Fanuc KAREL source: MSG_DISCO.kl

PROGRAM T
%NOLOCKGROUP
VAR
 v0 : STRING[40]
 v1 : INTEGER
BEGIN
 MSG_DISCO(v0, v1)
END T
